FUNCTION_BLOCK FB_RechazarPieza_SFC

VAR_IN_OUT
	TpoRechazador: TIME;
END_VAR

VAR_INPUT
    // SFC-Flags
    SFCPause: BOOL;
    SFCReset: BOOL;
    
    // Indicadores de sincronizacion
    Ack: BOOL := TRUE;
    Execute: BOOL;
    
    // Entradas
    RechazadorDetras : BOOL;
	RechazadorDelante : BOOL;
	RechazadorArriba : BOOL;
	RechazadorVacio : BOOL;
	PulsadorMarcha: BOOL;
END_VAR
VAR_OUTPUT
    // Indicadores de sincronizacion
    Done: BOOL;
    Ready: BOOL;
	Fallo: BOOL;

    // Salidas
    RechazadorAvanza : BOOL;
	RechazadorRetrocede : BOOL;
	RechazadorBaja : BOOL;
	RechazadorSucciona : BOOL;
END_VAR
VAR
END_VAR

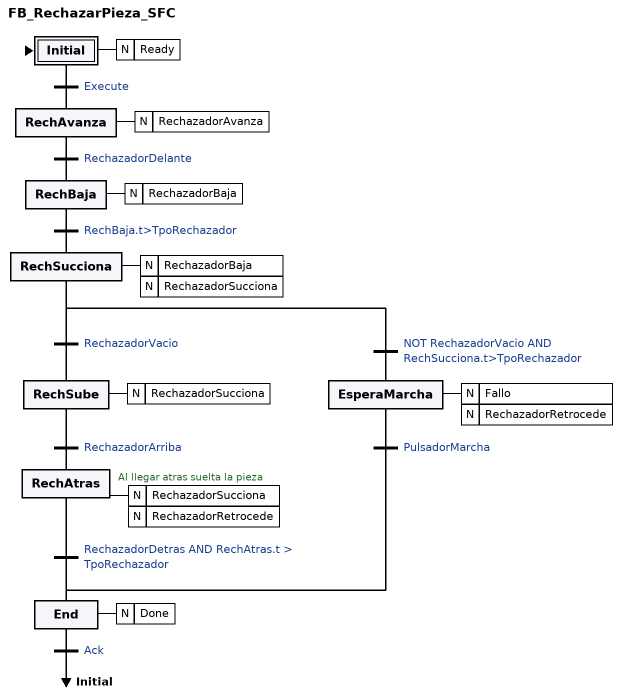
INITIAL_STEP Initial:
    Ready(N);
END_STEP
TRANSITION FROM Initial TO RechAvanza
    := Execute;
END_TRANSITION
STEP RechAvanza:
    RechazadorAvanza(N);
END_STEP
TRANSITION FROM RechAvanza TO RechBaja
    := RechazadorDelante;
END_TRANSITION
STEP RechBaja:
    RechazadorBaja(N);
END_STEP
TRANSITION FROM RechBaja TO RechSucciona
    := RechBaja.t>TpoRechazador;
END_TRANSITION
STEP RechSucciona:
    RechazadorBaja(N);
    RechazadorSucciona(N);
END_STEP
TRANSITION FROM RechSucciona TO RechSube
    := RechazadorVacio;
END_TRANSITION
STEP RechSube:
    RechazadorSucciona(N);
END_STEP
TRANSITION FROM RechSube TO RechAtras
    := RechazadorArriba;
END_TRANSITION
// Al llegar atras suelta la pieza
STEP RechAtras:
    RechazadorSucciona(N);
    RechazadorRetrocede(N);
END_STEP
TRANSITION FROM RechAtras TO End
    := RechazadorDetras AND RechAtras.t > TpoRechazador;
END_TRANSITION
TRANSITION FROM RechSucciona TO EsperaMarcha
    := NOT RechazadorVacio AND RechSucciona.t>TpoRechazador;
END_TRANSITION
STEP EsperaMarcha:
    Fallo(N);
    RechazadorRetrocede(N);
END_STEP
TRANSITION FROM EsperaMarcha TO End
    := PulsadorMarcha;
END_TRANSITION
STEP End:
    Done(N);
END_STEP
TRANSITION FROM End TO Initial
    := Ack;
END_TRANSITION

END_FUNCTION_BLOCK

(* stored: Version 1.1.0.1, ProductVersion 3.1.4024.12
   POU FB_RechazarPieza_SFC: Id {2f87a32f-15d5-4920-9713-8b43456c9444}, SpecialFunc None *)
